{attribute addProperty BoxType "EL3773-0000-0019"}
{attribute addProperty Id "U2_SamplesAT %I*ARRAY [0..9] OF INT16020"}
{attribute addProperty CRC "3561116077"}
{attribute addProperty SizeInBites "160"}
{attribute addProperty SizeInBytes "20"}
TYPE L2_Voltage_Samples_D44251AD :
STRUCT
	{attribute addProperty Name "U2_Samples"}
	U2_Samples AT %I* : ARRAY [0..9] OF INT;
END_STRUCT
END_TYPE

(* stored: Version 1.2.0.0, ProductVersion 3.1.4024.9
   DUT L2_Voltage_Samples_D44251AD: Id {20df92a3-4e5e-4df7-90e6-40a470c5fcdf} *)
